(* CODESYS project Passo-4.project

Project tree, tasks and I/O mapping:
  Device : CODESYS Control Win V3, 3S - Smart Software Solutions GmbH, order no. 305021, version 3.5.11.30
    application Application
      libraries: Standard, * (System)
      task MainTask (cyclic, interval t#20ms, priority 1) calls PLC_PRG
      program PLC_PRG [ST]
      Symbols
*)

// Device/Application/PLC_PRG
PROGRAM PLC_PRG
VAR
	DELAY:BOOL;
	//TIMERS
	TIMER: TON;
	//BOTOES
	START_BUTTON: BOOL;
	RESET: BOOL;
	EMERGENCY_BUTTON:BOOL;
	//SENSORES
	VISION_SENSOR: ARRAY[0..3] OF BOOL;
	MCBUSY: BOOL;
	
	REFLECTIVE1: BOOL;
	REFLECTIVE2:BOOL;
	DIFFUSE1:   ARRAY [1..2] OF BOOL;
	DIFFUSE2:   ARRAY [1..2] OF BOOL;
	DIFFUSEA: BOOL;
	DIFFUSEV: BOOL;
	DIFFUSEC: BOOL;
	//ATUADORES
	POSITIONER1: BOOL := 0;
	POSITIONER2: BOOL := 0;
	
	CINZA: BOOL;
	VERDE: BOOL;
	AZUL: BOOL;
	
	EMIT: BOOL;
	EMITTER_PART2: INT;
	EMIT2: BOOL := 0;
	
	ESTEIRA1: ARRAY [1..5] OF BOOL;
	ESTEIRA2: ARRAY [1..5] OF BOOL;
	ESTEIRAC: BOOL;
	ESTEIRAV: ARRAY [1..3] OF BOOL;
	ESTEIRAA: ARRAY [1..3] OF BOOL;
	//PICK & PLACE
	Z: REAL := 0;
	X: REAL := 2;//X: REAL := 1.1;
	Y: REAL := 0;
	GRAB: BOOL := 0;
	DETECTING: BOOL;
	//AUXILIARES
	PROGRESS_FLAG: WORD := 0;
	GRAB_FLAG: BOOL;
	PRODUZIR_LID: BOOL := TRUE;
	COUNT_AZUL: WORD := 0;
	COUNT_CINZA:WORD := 0;
	COUNT_VERDE:WORD := 0;
	COLOR_BUFFER: ARRAY[1..2] OF BYTE;
END_VAR

TIMER(IN:= DELAY, PT:= T#1S);
//RESET
IF RESET THEN
	Z := 0;
	X := 2;
	Y := 0;
	GRAB := FALSE;
	ESTEIRA1[1] := ESTEIRA1[2] := ESTEIRA1[3] := ESTEIRA1[4] := ESTEIRA1[5] := FALSE;
	ESTEIRA2[1] := ESTEIRA2[2] := ESTEIRA2[3] := ESTEIRA2[4] := ESTEIRA2[5] := FALSE;
	ESTEIRAA[1] := ESTEIRAA[2] := ESTEIRAA[3] := FALSE;
	ESTEIRAV[1] := ESTEIRAV[2] := ESTEIRAV[3] := FALSE;
	ESTEIRAC := FALSE; 
	EMIT := FALSE;
	EMIT2 := FALSE;
	GRAB_FLAG := FALSE;
	DELAY := FALSE;
	POSITIONER1 := FALSE;
	POSITIONER2 := FALSE;
	RESET := FALSE;
	PROGRESS_FLAG := 0;
	COUNT_CINZA := 0;
	COUNT_AZUL := 0;
	COUNT_VERDE := 0;
	COLOR_BUFFER[1] := 0;
	COLOR_BUFFER[2] := 0;
END_IF

//CONTROLANDO ESTEIRAS 
ESTEIRA1[1]  := EMIT := START_BUTTON AND (NOT DIFFUSE1[1]) AND (NOT MCBUSY) AND (NOT DIFFUSE1[2]);
ESTEIRA2[1] := EMIT2 := DIFFUSE1[1] AND (NOT DIFFUSE2[1]);

IF DIFFUSE1[2] THEN
	ESTEIRA1[2] := ESTEIRA1[3] := ESTEIRA1[4] := ESTEIRA1[5] := TRUE;
END_IF

IF DIFFUSE2[2] AND ESTEIRA1[2] THEN
	ESTEIRA2[2] := ESTEIRA2[3] := ESTEIRA2[4] := ESTEIRA2[5] := TRUE;
END_IF

IF PROGRESS_FLAG > 1 THEN
	ESTEIRA1[2] := ESTEIRA1[3] := ESTEIRA1[4] := ESTEIRA1[5] := FALSE;
	ESTEIRA2[2] := ESTEIRA2[3] := ESTEIRA2[4] := ESTEIRA2[5] := FALSE;
END_IF

IF DIFFUSEA THEN
	ESTEIRAA[1] := ESTEIRAA[2] := ESTEIRAA[3] := FALSE;
END_IF

IF DIFFUSEC THEN
	ESTEIRAC := FALSE;
END_IF

IF DIFFUSEV THEN
	ESTEIRAV[1] := ESTEIRAV[2] := ESTEIRAV[3] := FALSE;
END_IF

//USANDO SENSOR PRA DETECTAR COR DE OBTEJO
//Detectando a cor do objeto e gerando moldura correspondente
IF VISION_SENSOR[1] THEN
	EMITTER_PART2 := 64; CINZA := TRUE; VERDE := FALSE; AZUL := FALSE; //CINZA
	
ELSIF VISION_SENSOR[0] THEN
	EMITTER_PART2 := 16; CINZA := FALSE; VERDE := FALSE; AZUL := TRUE; //AZUL
	
ELSIF VISION_SENSOR[2] THEN
	EMITTER_PART2 := 32; CINZA := FALSE; VERDE := TRUE; AZUL := FALSE; //VERDE
END_IF

//Salvando a cor lida em um buffer, para que a próxima peça não sobreponha a anterior
IF VISION_SENSOR[0] OR VISION_SENSOR[1] OR VISION_SENSOR[2] THEN
	IF COLOR_BUFFER[1] = 0 THEN
		IF CINZA THEN
			COLOR_BUFFER[1] := 1;
		ELSIF VERDE THEN
			COLOR_BUFFER[1] := 2;
		ELSIF AZUL THEN
			COLOR_BUFFER[1] := 3;
		END_IF
	ELSE
		IF CINZA THEN
			COLOR_BUFFER[2] := 1;
		ELSIF VERDE THEN
			COLOR_BUFFER[2] := 2;
		ELSIF AZUL THEN
			COLOR_BUFFER[2] := 3;
		END_IF
	END_IF
END_IF

//CONTROLANDO PICK & PLACE
//PROGRESS = 1
IF NOT REFLECTIVE1 THEN
	PROGRESS_FLAG := 30; //Impedir que peças bases sejam acumuladas
END_IF

IF NOT REFLECTIVE2 THEN
	PROGRESS_FLAG := 1;
	DELAY := TRUE;
END_IF

//PROGRESS = 2
IF POSITIONER1 THEN
	DELAY:=TRUE;
END_IF

//PROGRESS = 3
IF DETECTING AND NOT GRAB_FLAG THEN
	GRAB_FLAG := TRUE;
	DELAY := TRUE;
END_IF

//PROGRESS = 4
IF GRAB_FLAG AND NOT DELAY THEN
	DELAY := TRUE;
END_IF

//PROGRESS = 5
IF PROGRESS_FLAG = 6 THEN
	DELAY := TRUE;
END_IF

IF Z = 3 THEN
	DELAY := TRUE;
END_IF

IF PROGRESS_FLAG = 9 AND NOT DELAY THEN
	DELAY := TRUE;
END_IF

IF TIMER.Q THEN
	DELAY := FALSE;
	IF PROGRESS_FLAG = 9 THEN
		IF COUNT_CINZA > 1 THEN
			ESTEIRAC := TRUE; 
			COUNT_CINZA := 0;
		ELSIF COUNT_AZUL > 1 THEN
			ESTEIRAA[1] := ESTEIRAA[2] := ESTEIRAA[3] := TRUE;
			COUNT_AZUL := 0; 
		ELSIF COUNT_VERDE > 1 THEN
			ESTEIRAV[1] := ESTEIRAV[2] := ESTEIRAV[3] := TRUE;
			COUNT_VERDE := 0; 
		END_IF
		COLOR_BUFFER[1] := COLOR_BUFFER[2];
			Z := 0;
			X := 2;
			Y := 0;
			GRAB := FALSE;
			GRAB_FLAG := FALSE;
			PROGRESS_FLAG := 0;
		
	ELSIF PROGRESS_FLAG = 8 THEN
		GRAB := FALSE;
		PROGRESS_FLAG := 9;
		
	ELSIF PROGRESS_FLAG = 7 THEN
		IF COLOR_BUFFER[1] = 1 THEN //É CINZA
			X := 5;
			Y := 10;
			COUNT_CINZA := COUNT_CINZA + 1;

		ELSIF COLOR_BUFFER[1] = 3 THEN //É AZUL
			X := 0;
			Y := 7;
			COUNT_AZUL := COUNT_AZUL + 1;
		ELSIF COLOR_BUFFER[1] = 2 THEN //É VERDE
			X := 10;
			Y := 7;
			COUNT_VERDE := COUNT_VERDE + 1;
		END_IF
		PROGRESS_FLAG := 8;
		
	ELSIF PROGRESS_FLAG = 6 THEN
		Z := 0;
		PROGRESS_FLAG := 7;
		
	ELSIF PROGRESS_FLAG = 5 THEN
		Z := 8.2;
		PROGRESS_FLAG := 6;
	
	ELSIF PROGRESS_FLAG = 4 THEN
		X := 7.3;
		PROGRESS_FLAG := 5;
		
	ELSIF PROGRESS_FLAG = 3 THEN
		Z := 3;
		PROGRESS_FLAG := 4;
		
	ELSIF PROGRESS_FLAG = 2 THEN
		POSITIONER1 := FALSE;
		POSITIONER2 := FALSE;
		GRAB := TRUE;
		Z := 8.2;
		PROGRESS_FLAG := 3;
		
	ELSIF PROGRESS_FLAG = 1 THEN
		POSITIONER1 := TRUE;
		POSITIONER2 := TRUE;
		PROGRESS_FLAG := 2;
	END_IF
END_IF

END_PROGRAM
